PROGRAM MAIN
VAR
	systemOk				AT %I* :BOOL;
	estopPressed			AT %I* :BOOL;
	safeGroupErrorReset  	AT %Q* :BOOL;
	doorUnlock_But		 	AT %Q* :BOOL;	
	
	SafetyResetPulse				: TP;
	
	Control							: fbControl;
	InfeedConveyor					: fbInConveyor;
	HousingDelivery					: fbHousingDelivery;
	InsertPlacing					: fbInsertPlacing;
	Handling						: fbHandling;
	Pressing						: fbPressing;
	
END_VAR

doorUnlock_But := HMI.DoorUnlockCmd;
//gpb.estopOk := systemOk;

//===============================================================================================
// Safety reset at system startup
//===============================================================================================
SafetyResetPulse(IN:=TRUE, PT:= T#500MS , Q=>safeGroupErrorReset , ET=> );



//===============================================================================================
// Machine modes and status indication 
//===============================================================================================

Control(
	SafetyOk:= SystemOk,
	ResetCompleted := TRUE,
	ResetCmd=> , 
	AutoCycle=> , 
	ManualMode=> , 
	DoorUnlockCmd=> );

//===============================================================================================
// Infeed conveyor control  
//===============================================================================================

InfeedConveyor(
	SafetyOk:= , 
	ResetCmd:= , 
	AutoCycle:= , 
	ManualCmd:= , 
	ResetCompleted=> );


	
	
//===============================================================================================
// Fitting station process control  
//===============================================================================================

HousingDelivery(
	SafetyOk:= , 
	ResetCmd:= , 
	AutoCycle:= , 
	ManualCmd:= , 
	ResetCompleted=> );
	
InsertPlacing(
	SafetyOk:= , 
	ResetCmd:= , 
	AutoCycle:= , 
	ManualCmd:= , 
	ResetCompleted=> );	

	
//===============================================================================================
// Pressing station process control  
//===============================================================================================	


Handling(
	SafetyOk:= , 
	ResetCmd:= , 
	AutoCycle:= , 
	ManualCmd:= , 
	ResetCompleted=> );


Pressing(
	SafetyOk:= , 
	ResetCmd:= , 
	AutoCycle:= , 
	ManualCmd:= , 
	ResetCompleted=> );

END_PROGRAM

(* stored: Version 1.1.0.1, ProductVersion 3.1.4022.18
   POU MAIN: Id {21da2244-018d-444a-95bb-341d673e2187}, SpecialFunc None *)
